PROGRAM Analog_Speed
VAR
	fScaledSpeed				:DINT;
END_VAR

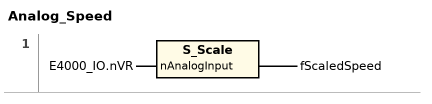
// NETWORK 1
fScaledSpeed := S_Scale(nAnalogInput := E4000_IO.nVR);

END_PROGRAM

(* stored: Version 1.1.0.1, ProductVersion 3.1.4024.0
   POU Analog_Speed: Id {ad069b50-b61e-4052-b5a2-03a1d45702ac}, SpecialFunc None *)
